Fanuc KAREL source: ka00133.KL

PROGRAM KA00133
%NOLOCKGROUP
VAR
SRC : ARRAY[2] OF SHORT
DST:INTEGER
BEGIN
SRC[1]=2
DST=SRC[1]
END KA00133
